FUNCTION_BLOCK Test_AddEventHandler_ChecksInterfaceSupported EXTENDS TUnitTestbase
VAR_INPUT
END_VAR
VAR_OUTPUT
END_VAR
VAR
    TestEvent : TTestEvent;
    TestEventHandler : TUnsupportedEventHandler;
END_VAR

METHOD  Execute
TestEvent.ClearEventHandlers().AddEventHandler(TestEventHandler); // should trigger an error message

Assertion.AssertEquals_DINT(
    Expected := 0,
    Actual   := TestEvent.EventHandlers.Count,
    ObjectName := _TestName,
    VariableName  := 'TestEvent.EventHandlers.Count');

_TestFinished := TRUE;
END_METHOD

END_FUNCTION_BLOCK

(* stored: Version 1.1.0.1, ProductVersion 3.1.4024.3
   POU Test_AddEventHandler_ChecksInterfaceSupported: Id {a9f1d7f7-cf42-4f58-85a0-dd9941b77fb1}, SpecialFunc None
   Method Execute: Id {dd4a142a-404c-4e57-aef9-46db63b892c9} *)
